KUKA KRL program: cadmatch_detect.src, cadmatch_detect.dat

--- cadmatch_detect.src ---
&ACCESS RVO
&REL 116
&PARAM EDITMASK = *
&PARAM TEMPLATE = C:\KRC\Roboter\Template\vorgabe
&PARAM DISKPATH = KRC:\R1\Program
DEF cadmatch_detect( )

   DECL CHAR serviceName[32]
   DECL EKI_Status RET
   DECL FRAME CADMatchingPose

   ;FOLD INI;%{PE}
      ;FOLD BASISTECH INI
         GLOBAL INTERRUPT DECL 3 WHEN $STOPMESS==TRUE DO IR_STOPM ( )
         INTERRUPT ON 3
         BAS (#INITMOV,0 )
      ;ENDFOLD (BASISTECH INI)
      ;FOLD USER INI
         ;Make your modifications here

      ;ENDFOLD (USER INI)
   ;ENDFOLD (INI)

   INTERRUPT DECL 89 WHEN $FLAG[998] DO RC_NOTIFYRECEIVED(1, 998)
   INTERRUPT ON 89

   ;FOLD SPTP HOME Vel=100 % DEFAULT;%{PE}%MKUKATPBASIS,%CSPLINE,%VSPTP_SB,%P 1:SPTP_SB, 2:HOME, 3:, 5:100, 7:DEFAULT
      SPTP XHOME WITH $VEL_AXIS[1]= SVEL_JOINT( 100), $TOOL= STOOL2( FHOME), $BASE= SBASE( FHOME.BASE_NO),$IPO_MODE= SIPO_MODE( FHOME.IPO_FRAME), $LOAD= SLOAD( FHOME.TOOL_NO), $ACC_AXIS[1]= SACC_JOINT( PDEFAULT), $GEAR_JERK[1]= SGEAR_JERK( PDEFAULT)
   ;ENDFOLD

   ; Init cadmatch module and open connection to rc_cube
   RC_START()
   $FLAG[1] = FALSE
   RC_SETMSG("Start")
   serviceName[] = "rc_cadmatch-detect_object"
   RC_INIT(serviceName[])
   RC_OPENCONNECTION(serviceName[])

   LOOP

      ; Reset vision results
      WAIT SEC 0
      ResetDetectedItems()

      ;****************************************
      ; Mandatory application parameters:
      ; ---------------------------------
      ; Template ID (Part) [Default: "Template_1"]
      ; Pose Frame, sensor or robot (external) [Default: "external"]
      ;****************************************
      RET = EKI_SetString(serviceName[], "req/args/template_id", "Template_1")
      RET = EKI_SetString(serviceName[], "req/args/pose_frame", "external")

      ;****************************************
      ; Optional application parameters:
      ; --------------------------------
      ; Load Carrier ID (Box) [Default: "LoadCarrier_1"]
      ; Region of Interest ID [Default: "RegionOfInterest_1"]
      ; Gripper ID [Default: "Gripper_1"]
      ; Offset pre Pick for collision detection [Default: X 0.0, Y 0.0, Z -0.5]
      ; LC Box, if load carrier should be configured externally [Default: X 0.0, Y 0.0, Z 0.0]
      ; LC Pose, if load carrier should be configured externally [Default: X 0.0, Y 0.0, Z 0.0, A 0.0, B 0.0, C 0.0]
      ; Robot Pose, only relevant for robot mounted sensor [Default: X 0.0, Y 0.0, Z 0.0, A 0.0, B 0.0, C 0.0]
      ;****************************************
      RET = EKI_SetString(serviceName[], "req/args/load_carrier_id", "LoadCarrier_1")
      RET = EKI_SetString(serviceName[], "req/args/region_of_interest_id", "RegionOfInterest_1")
      RET = EKI_SetString(serviceName[], "req/args/collision_detection/@gripper_id", "Gripper_1")
      RET = EKI_SetReal(serviceName[], "req/args/collision_detection/pre_grasp_offset/@x", 0.0)
      RET = EKI_SetReal(serviceName[], "req/args/collision_detection/pre_grasp_offset/@y", 0.0)
      RET = EKI_SetReal(serviceName[], "req/args/collision_detection/pre_grasp_offset/@z", -0.5)
      ;RET = EKI_SetReal(serviceName[], "req/args/load_carrier_compartment/box/@x ", 0.0)
      ;RET = EKI_SetReal(serviceName[], "req/args/load_carrier_compartment/box/@y ", 0.0)
      ;RET = EKI_SetReal(serviceName[], "req/args/load_carrier_compartment/box/@z ", 0.0)
      ;RET = EKI_SetReal(serviceName[], "req/args/load_carrier_compartment/pose/@X ", 0.0)
      ;RET = EKI_SetReal(serviceName[], "req/args/load_carrier_compartment/pose/@Y ", 0.0)
      ;RET = EKI_SetReal(serviceName[], "req/args/load_carrier_compartment/pose/@Z ", 0.0)
      ;RET = EKI_SetReal(serviceName[], "req/args/load_carrier_compartment/pose/@A ", 0.0)
      ;RET = EKI_SetReal(serviceName[], "req/args/load_carrier_compartment/pose/@B ", 0.0)
      ;RET = EKI_SetReal(serviceName[], "req/args/load_carrier_compartment/pose/@C ", 0.0)
      ;RET = EKI_SetReal(serviceName[], "req/args/robot_pose/@X", 0.0)
      ;RET = EKI_SetReal(serviceName[], "req/args/robot_pose/@Y", 0.0)
      ;RET = EKI_SetReal(serviceName[], "req/args/robot_pose/@Z", 0.0)
      ;RET = EKI_SetReal(serviceName[], "req/args/robot_pose/@A", 0.0)
      ;RET = EKI_SetReal(serviceName[], "req/args/robot_pose/@B", 0.0)
      ;RET = EKI_SetReal(serviceName[], "req/args/robot_pose/@C", 0.0)

      ; Send trigger and wait for vision results
      RET = EKI_Send(serviceName[], "req")
      RC_WAITFORRESULT(1)
      RC_READRESULT(serviceName[])

      ; Error handling
      IF (RETURNCODE.VALUE < 0) THEN
         RC_SETMSG("Execution failed")
         RC_SETMSG(RETURNCODE.MSG[])
         HALT
      ENDIF

      ; No CAD matching result found
      IF NOT(CheckDetectedItem(1)) THEN
         MsgQuit("No CAD matchin vision result found","RC")
         HALT
      ENDIF

      ;Calculate pick position on first detected part
      CADMatchingPose=DETECTEDITEMS[1]
      xP1 = CADMatchingPose

      ; Pre pick position
      ;FOLD SPTP P2 CONT Vel=100 % PDAT4 Tool[2]:Magnet Base[0] ;%{PE}
         ;FOLD Parameters ;%{h}
            ;Params IlfProvider=kukaroboter.basistech.inlineforms.movement.spline; Kuka.IsGlobalPoint=False; Kuka.PointName=P2; Kuka.BlendingEnabled=True; Kuka.MoveDataPtpName=PDAT4; Kuka.VelocityPtp=100; Kuka.VelocityFieldEnabled=True; Kuka.ColDetectFieldEnabled=True; Kuka.CurrentCDSetIndex=0; Kuka.MovementParameterFieldEnabled=True; IlfCommand=SPTP
         ;ENDFOLD
         SPTP XP2 WITH $VEL_AXIS[1] = SVEL_JOINT(100.0), $TOOL = STOOL2(FP2), $BASE = SBASE(FP2.BASE_NO), $IPO_MODE = SIPO_MODE(FP2.IPO_FRAME), $LOAD = SLOAD(FP2.TOOL_NO), $ACC_AXIS[1] = SACC_JOINT(PPDAT4), $APO = SAPO_PTP(PPDAT4), $GEAR_JERK[1] = SGEAR_JERK(PPDAT4), $COLLMON_TOL_PRO[1] = USE_CM_PRO_VALUES(0) C_Spl
      ;ENDFOLD

      ; Pick position
      ;FOLD LIN P1 Vel=0.2 m/s CPDAT1 Tool[2]:Magnet Base[0] ;%{PE}
         ;FOLD Parameters ;%{h}
            ;Params IlfProvider=kukaroboter.basistech.inlineforms.movement.old; Kuka.IsGlobalPoint=False; Kuka.PointName=P1; Kuka.BlendingEnabled=False; Kuka.MoveDataName=CPDAT1; Kuka.VelocityPath=0.2; Kuka.CurrentCDSetIndex=0; Kuka.MovementParameterFieldEnabled=True; IlfCommand=LIN
         ;ENDFOLD
         $BWDSTART = FALSE
         LDAT_ACT = LCPDAT1
         FDAT_ACT = FP1
         BAS(#CP_PARAMS, 0.2)
         SET_CD_PARAMS (0)
         LIN XP1
      ;ENDFOLD

      ; Post pick position
      ;FOLD LIN P2 CONT Vel=2 m/s CPDAT3 Tool[2]:Magnet Base[0] ;%{PE}
         ;FOLD Parameters ;%{h}
            ;Params IlfProvider=kukaroboter.basistech.inlineforms.movement.old; Kuka.IsGlobalPoint=False; Kuka.PointName=P2; Kuka.BlendingEnabled=True; Kuka.MoveDataName=CPDAT3; Kuka.VelocityPath=2; Kuka.CurrentCDSetIndex=0; Kuka.MovementParameterFieldEnabled=True; IlfCommand=LIN
         ;ENDFOLD
         $BWDSTART = FALSE
         LDAT_ACT = LCPDAT3
         FDAT_ACT = FP2
         BAS(#CP_PARAMS, 2.0)
         SET_CD_PARAMS (0)
         LIN XP2 C_Dis C_Dis
      ;ENDFOLD

      RC_SETMSG("Finish")

      ; Place position
      ;FOLD SPTP P3 Vel=100 % PDAT3 Tool[2] Base[0] ;%{PE}
         ;FOLD Parameters ;%{h}
            ;Params IlfProvider=kukaroboter.basistech.inlineforms.movement.spline; Kuka.IsGlobalPoint=False; Kuka.PointName=P3; Kuka.BlendingEnabled=False; Kuka.MoveDataPtpName=PDAT3; Kuka.VelocityPtp=100; Kuka.VelocityFieldEnabled=True; Kuka.ColDetectFieldEnabled=True; Kuka.CurrentCDSetIndex=0; Kuka.MovementParameterFieldEnabled=True; IlfCommand=SPTP
         ;ENDFOLD
         SPTP XP3 WITH $VEL_AXIS[1] = SVEL_JOINT(100.0), $TOOL = STOOL2(FP3), $BASE = SBASE(FP3.BASE_NO), $IPO_MODE = SIPO_MODE(FP3.IPO_FRAME), $LOAD = SLOAD(FP3.TOOL_NO), $ACC_AXIS[1] = SACC_JOINT(PPDAT3), $APO = SAPO_PTP(PPDAT3), $GEAR_JERK[1] = SGEAR_JERK(PPDAT3), $COLLMON_TOL_PRO[1] = USE_CM_PRO_VALUES(0)
      ;ENDFOLD

      ;FOLD SPTP HOME Vel=100 % DEFAULT;%{PE}%MKUKATPBASIS,%CSPLINE,%VSPTP_SB,%P 1:SPTP_SB, 2:HOME, 3:, 5:100, 7:DEFAULT
         SPTP XHOME WITH $VEL_AXIS[1]= SVEL_JOINT( 100), $TOOL= STOOL2( FHOME), $BASE= SBASE( FHOME.BASE_NO),$IPO_MODE= SIPO_MODE( FHOME.IPO_FRAME), $LOAD= SLOAD( FHOME.TOOL_NO), $ACC_AXIS[1]= SACC_JOINT( PDEFAULT), $GEAR_JERK[1]= SGEAR_JERK( PDEFAULT)
      ;ENDFOLD

   ENDLOOP

   RC_STOP()
   RC_CLOSECONNECTION(serviceName[], "req")

END

;FOLD RC_SETMSG
   DEF RC_SETMSG(msg[]:IN)
      DECL CHAR msg[]
      DECL KrlMsgPar_T params[3]
      RC_SETMSG_PARAM(msg[], params[])
   END

;ENDFOLD (RC_SETMSG)

;FOLD RC_SETMSG_PARAM
DEF RC_SETMSG_PARAM(msg[]:IN, params:OUT)
  DECL CHAR msg[]
  DECL KrlMsgPar_T params[]

  DECL KrlMsg_T name
  DECL KrlMsgOpt_T options
  DECL INT Handle, len, count
  DECL EKrlMsgType Type

  name={modul[] "RC", nr 1, msg_txt[] " "}

  Type=#notify

  len=STRLEN(msg[])
  IF len>0 THEN
    IF len>80 THEN
      len=80
    ENDIF
    FOR count=1 TO len
      name.msg_txt[count]=msg[count]
    ENDFOR
  ELSE
    name.msg_txt[]="parameter msg[] is missing"
  ENDIF

  Handle=Set_KrlMsg(Type, name, params[], options)
END
;ENDFOLD (RC_SETMSG_PARAM)

;FOLD RC_INIT
   DEF RC_INIT(configFileName[]:IN)
      DECL CHAR configFileName[]
      DECL EKI_Status RET
      RET=EKI_INIT(configFileName[])
   END

;ENDFOLD (RC_INIT)

;FOLD RC_OPENCONNECTION
   DEF RC_OPENCONNECTION(configFileName[]:IN)
      DECL CHAR configFileName[]
      DECL EKI_Status RET
      RET=EKI_Open(configFileName[])
      EKI_CHECK(RET,#Quit)
   END

;ENDFOLD (RC_OPENCONNECTION)

;FOLD RC_CLOSECONNECTION
   DEF RC_CLOSECONNECTION(configFileName[]:IN, strPlace[]:IN)
      DECL CHAR configFileName[]
      DECL CHAR strPlace[]
      DECL EKI_Status RET
      WAIT SEC 0
      RET=EKI_Close(configFileName[])
      RET=EKI_ClearBuffer(configFileName[], strPlace[])
   END
;ENDFOLD (RC_CLOSECONNECTION)

;FOLD RC_WAITFORRESULT
   DEF RC_WAITFORRESULT(WaitFlag:IN)
      DECL INT WaitFlag

      WAIT FOR $FLAG[WaitFlag] OR NOT $FLAG[RCEkiAliveFlagNo]

      ;Eki-connection has been closed

      IF(NOT $FLAG[RCEkiAliveFlagNo]) THEN
         RC_SETMSG("EKI connection lost")
      ENDIF

      $FLAG[WaitFlag] = FALSE
      WAIT SEC 0
   END

;ENDFOLD (RC_WAITFORRESULT)

;FOLD RC_NOTIFYRECEIVED
   DEF RC_NOTIFYRECEIVED(WAITFLAG:IN, EOFRESULFLAG:IN)
      DECL INT WAITFLAG
      DECL INT EOFRESULFLAG
      $FLAG[EOFRESULFLAG]=FALSE
      $FLAG[WAITFLAG]=TRUE
   END

;ENDFOLD (RC_NOTIFYRECEIVED)

;FOLD RC_READRESULT
   DEF RC_READRESULT(configFileName[]:IN)
      DECL CHAR configFileName[]
      DECL RETURNCODE_T RESULT
      DECL EKI_STATUS RET
      DECL INT j
      DECL FRAME POSE

      POSE = POSE_IDENT

      RESULT={VALUE 0, MSG[] "0"}

      ;Standard Kommunikation fuer Fehlercode
      RET = EKI_GetInt(configFileName[], "res/return_code/@value", RESULT.VALUE)
      RET = EKI_GetString(configFileName[], "res/return_code/@message", RESULT.MSG[])
      RETURNCODE = RESULT

      ;Kopieren der Anzahl an Greifpositionen
      RET = EKI_CheckBuffer(configFileName[], "res/grasps/le/id")
      NUMDETECTEDITEMS = RET.Buff

      ;Kopieren aller Greifpositionen
      for j=1 to NUMDETECTEDITEMS

         RET = EKI_GetFrame(configFileName[], "res/grasps/le/pose", POSE)
         DETECTEDITEMS[j] = POSE

      endfor

      RET = EKI_ClearBuffer(configFileName[], "res")
   END

;ENDFOLD (RC_READRESULT)

;FOLD RC_START
   DEF RC_START()

      DECL CHAR serviceName[32]
      DECL EKI_Status RET

      ; Init
      $FLAG[1] = FALSE
      RC_SETMSG("Start")
      serviceName[] = "rc_cadmatch-start"

      ; Open connection
      RC_INIT(serviceName[])
      RC_OPENCONNECTION(serviceName[])

      ; Trigger vision
      RET = EKI_Send(serviceName[], "req")

      ; Wait for vision result
      RC_WAITFORRESULT(1)

      ; Close connection
      RC_CLOSECONNECTION(serviceName[], "req")

   END

;ENDFOLD (RC_START)

;FOLD RC_STOP
   DEF RC_STOP()

      DECL CHAR serviceName[32]
      DECL EKI_Status RET

      ; Init
      $FLAG[1] = FALSE
      RC_SETMSG("Stop")
      serviceName[] = "rc_cadmatch-stop"

      ; Open connection
      RC_INIT(serviceName[])
      RC_OPENCONNECTION(serviceName[])

      ; Trigger vision
      RET = EKI_Send(serviceName[], "req")

      ; Wait for vision result
      RC_WAITFORRESULT(1)

      ; Close connection
      RC_CLOSECONNECTION(serviceName[], "req")

   END

;ENDFOLD (RC_STOP)

;FOLD (ResetDetectedItems)
   DEF ResetDetectedItems()
      DECL INT I

      FOR I = 1 TO 32 STEP 1
         DETECTEDITEMS[I]=$NULLFRAME
      ENDFOR
   END

;ENDFOLD (ResetDetectedItems)

;FOLD CheckDetectedItem
   DEFFCT BOOL CheckDetectedItem(Index:IN)
      DECL INT Index
      DECL KrlMsgPar_T par[3]

      IF (DETECTEDITEMS[Index].X == 0) AND (DETECTEDITEMS[Index].Y == 0) AND (DETECTEDITEMS[Index].Z == 0) AND (DETECTEDITEMS[Index].A == 0) AND (DETECTEDITEMS[Index].B == 0) AND (DETECTEDITEMS[Index].C ==0) THEN
         RETURN FALSE
      ELSE
         ;Meldung CAD MAtching Position
         par[1] = {par_type #value, par_real 0}
         par[1].par_real = DETECTEDITEMS[1].X
         par[2] = {par_type #value, par_real 0}
         par[2].par_real = DETECTEDITEMS[1].Y
         par[3] = {par_type #value, par_real 0}
         par[3].par_real = DETECTEDITEMS[1].Z
         RC_SETMSG_PARAM("CAD Matching Pose: X: %1, Y: %2, Z: %3", par[])
         RETURN TRUE
      ENDIF

   ENDFCT

;ENDFOLD (CheckDetectedItem)

--- cadmatch_detect.dat ---
&ACCESS RVP
&REL 116
&PARAM EDITMASK = *
&PARAM TEMPLATE = C:\KRC\Roboter\Template\vorgabe
&PARAM DISKPATH = KRC:\R1\Program
DEFDAT  CADMATCH_DETECT
;FOLD EXTERNAL DECLARATIONS;%{PE}%MKUKATPBASIS,%CEXT,%VCOMMON,%P
;FOLD BASISTECH EXT;%{PE}%MKUKATPBASIS,%CEXT,%VEXT,%P
EXT  BAS (BAS_COMMAND  :IN,REAL  :IN )
DECL INT SUCCESS
;ENDFOLD (BASISTECH EXT)
;FOLD USER EXT;%{E}%MKUKATPUSER,%CEXT,%VEXT,%P
;Make your modifications here
STRUC RETURNCODE_T INT VALUE,CHAR MSG[512]

DECL RETURNCODE_T RETURNCODE
DECL FRAME DETECTEDITEMS[32]
DECL INT NUMDETECTEDITEMS

DECL FRAME POSE_IDENT={X 0.0,Y 0.0,Z 0.0,A 0.0,B 0.0,C 0.0}

DECL INT RCEkiAliveFlagNo=997
;ENDFOLD (USER EXT)
;ENDFOLD (EXTERNAL DECLARATIONS)
DECL E6POS XP1={X 906.420837,Y 844.301514,Z -737.483765,A 109.228287,B 4.50301743,C 157.962234}
DECL FDAT FP1={TOOL_NO 2,BASE_NO 0,IPO_FRAME #BASE,POINT2[] " "}
DECL PDAT PPDAT1={VEL 100.000,ACC 100.000,APO_DIST 100.000,APO_MODE #CPTP,GEAR_JERK 50.0000,EXAX_IGN 0}
DECL MODULEPARAM_T LAST_TP_PARAMS={PARAMS[] "Kuka.VelocityFieldEnabled=True; Kuka.MovementParameterFieldEnabled=True; Kuka.PointName=P1; Kuka.FrameData.base_no=0; Kuka.FrameData.tool_no=2; Kuka.FrameData.ipo_frame=#BASE; Kuka.isglobalpoint=False; Kuka.MoveDataPtpName=PDAT6; Kuka.MovementDataPdat.apo_mode=#CDIS; Kuka.MovementDataPdat.apo_dist=20; Kuka.MovementData.vel=0.2; Kuka.MovementData.acc=100; Kuka.MovementData.gear_jerk=50; Kuka.MovementData.exax_ign=0; Kuka.VelocityPtp=100; Kuka.BlendingEnabled=False; Kuka.CurrentCDSetIndex=0; Kuka.FrameData.point2=; Kuka.ColDetectFieldEnabled=True; Kuka.IsAngleEnabled=False; Kuka.APXEnabled=False; Kuka.MoveDataName=CPDAT1; Kuka.MovementData.cb={AUX_PT {ORI #CONSIDER,E1 #CONSIDER,E2 #CONSIDER,E3 #CONSIDER,E4 #CONSIDER,E5 #CONSIDER,E6 #CONSIDER},TARGET_PT {ORI #INTERPOLATE,E1 #INTERPOLATE,E2 #INTERPOLATE,E3 #INTERPOLATE,E4 #INTERPOLATE,E5 #INTERPOLATE,E6 #INTERPOLATE}}; Kuka.MovementData.apo_fac=50; Kuka.MovementData.apo_dist=500; Kuka.MovementData.axis_acc=100; Kuka.MovementData.axis_vel=100; Kuka.MovementData.circ_typ=#BASE; Kuka.MovementData.jerk_fac=50; Kuka.MovementData.ori_typ=#VAR; Kuka.VelocityPath=0.2                  "}
DECL E6POS XP2={X 920.760376,Y 742.115417,Z -30.3186913,A 88.4895859,B 1.18707442,C -177.679535,S 2,T 43,E1 0.0,E2 0.0,E3 0.0,E4 0.0,E5 0.0,E6 0.0}
DECL FDAT FP2={TOOL_NO 2,BASE_NO 0,IPO_FRAME #BASE,POINT2[] " "}
DECL PDAT PPDAT2={VEL 100.000,ACC 100.000,APO_DIST 100.000,APO_MODE #CDIS,GEAR_JERK 100.000,EXAX_IGN 0}
DECL E6POS XP3={X 158.706436,Y 984.351685,Z 393.467163,A 88.5150757,B 1.08440256,C -177.713486,S 2,T 43,E1 0.0,E2 0.0,E3 0.0,E4 0.0,E5 0.0,E6 0.0}
DECL FDAT FP3={TOOL_NO 2,BASE_NO 0,IPO_FRAME #BASE,POINT2[] " "}
DECL PDAT PPDAT3={VEL 100.000,ACC 100.000,APO_DIST 100.000,APO_MODE #CDIS,GEAR_JERK 100.000,EXAX_IGN 0}
DECL LDAT LCPDAT1={VEL 0.200000,ACC 100.000,APO_DIST 500.000,APO_FAC 50.0000,AXIS_VEL 100.000,AXIS_ACC 100.000,ORI_TYP #VAR,CIRC_TYP #BASE,JERK_FAC 50.0000,GEAR_JERK 100.000,EXAX_IGN 0,CB {AUX_PT {ORI #CONSIDER,E1 #CONSIDER,E2 #CONSIDER,E3 #CONSIDER,E4 #CONSIDER,E5 #CONSIDER,E6 #CONSIDER},TARGET_PT {ORI #INTERPOLATE,E1 #INTERPOLATE,E2 #INTERPOLATE,E3 #INTERPOLATE,E4 #INTERPOLATE,E5 #INTERPOLATE,E6 #INTERPOLATE}}}
DECL LDAT LCPDAT2={VEL 2.00000,ACC 100.000,APO_DIST 500.000,APO_FAC 50.0000,AXIS_VEL 100.000,AXIS_ACC 100.000,ORI_TYP #VAR,CIRC_TYP #BASE,JERK_FAC 50.0000,GEAR_JERK 100.000,EXAX_IGN 0,CB {AUX_PT {ORI #CONSIDER,E1 #CONSIDER,E2 #CONSIDER,E3 #CONSIDER,E4 #CONSIDER,E5 #CONSIDER,E6 #CONSIDER},TARGET_PT {ORI #INTERPOLATE,E1 #INTERPOLATE,E2 #INTERPOLATE,E3 #INTERPOLATE,E4 #INTERPOLATE,E5 #INTERPOLATE,E6 #INTERPOLATE}}}
DECL PDAT PPDAT4={VEL 100.000,ACC 100.000,APO_DIST 20.0000,APO_MODE #CDIS,GEAR_JERK 100.000,EXAX_IGN 0}
DECL LDAT LCPDAT3={VEL 2.00000,ACC 100.000,APO_DIST 100.000,APO_FAC 50.0000,AXIS_VEL 100.000,AXIS_ACC 100.000,ORI_TYP #VAR,CIRC_TYP #BASE,JERK_FAC 50.0000,GEAR_JERK 100.000,EXAX_IGN 0,CB {AUX_PT {ORI #CONSIDER,E1 #CONSIDER,E2 #CONSIDER,E3 #CONSIDER,E4 #CONSIDER,E5 #CONSIDER,E6 #CONSIDER},TARGET_PT {ORI #INTERPOLATE,E1 #INTERPOLATE,E2 #INTERPOLATE,E3 #INTERPOLATE,E4 #INTERPOLATE,E5 #INTERPOLATE,E6 #INTERPOLATE}}}
DECL E6POS XH1={X 379.196655,Y 517.991699,Z 210.714554,A 88.4916,B 1.17288554,C -177.670990,S 2,T 43,E1 0.0,E2 0.0,E3 0.0,E4 0.0,E5 0.0,E6 0.0}
DECL FDAT FH1={TOOL_NO 2,BASE_NO 0,IPO_FRAME #BASE,POINT2[] " "}
DECL PDAT PPDAT5={VEL 100.000,ACC 100.000,APO_DIST 20.0000,APO_MODE #CDIS,GEAR_JERK 100.000,EXAX_IGN 0}
DECL PDAT PPDAT6={VEL 100.000,ACC 100.000,APO_DIST 20.0000,APO_MODE #CDIS,GEAR_JERK 100.000,EXAX_IGN 0}
ENDDAT
